// Mitsubishi GX Works2 project: auto0917   PLC: Q02/Q02H

PROGRAM MAIN
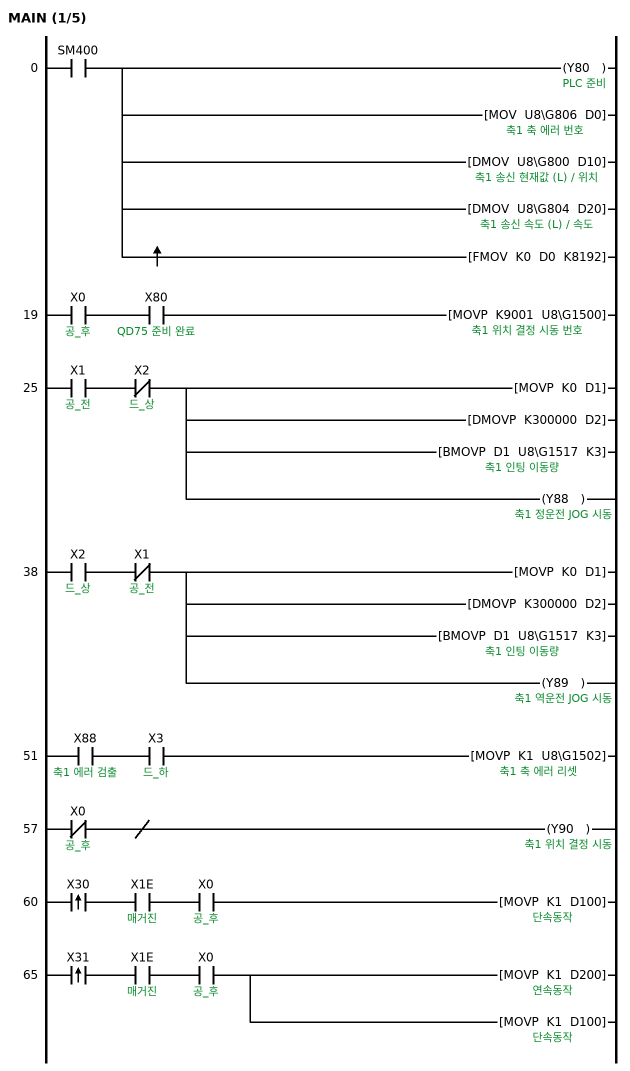
0     LD      SM400
      OUT     Y80  ; PLC 준비
      MOV     U8\G806 D0  ; 축1 축 에러 번호
      DMOV    U8\G800 D10  ; 축1 송신 현재값 (L) / 위치
      DMOV    U8\G804 D20  ; 축1 송신 속도 (L) / 속도
      MEP
      FMOV    K0 D0 K8192
19    LD      X0  ; 공_후
      AND     X80  ; QD75 준비 완료
      MOVP    K9001 U8\G1500  ; 축1 위치 결정 시동 번호
25    LD      X1  ; 공_전
      ANI     X2  ; 드_상
      MOVP    K0 D1
      DMOVP   K300000 D2
      BMOVP   D1 U8\G1517 K3  ; 축1 인팅 이동량
      OUT     Y88  ; 축1 정운전 JOG 시동
38    LD      X2  ; 드_상
      ANI     X1  ; 공_전
      MOVP    K0 D1
      DMOVP   K300000 D2
      BMOVP   D1 U8\G1517 K3
      OUT     Y89  ; 축1 역운전 JOG 시동
51    LD      X88  ; 축1 에러 검출
      AND     X3  ; 드_하
      MOVP    K1 U8\G1502  ; 축1 축 에러 리셋
57    LDI     X0  ; 공_후
      INV
      OUT     Y90  ; 축1 위치 결정 시동
60    LDP     X30
      AND     X1E  ; 매거진
      AND     X0  ; 공_후
      MOVP    K1 D100  ; 단속동작
65    LDP     X31
      AND     X1E  ; 매거진
      AND     X0  ; 공_후
      MOVP    K1 D200  ; 연속동작
      MOVP    K1 D100
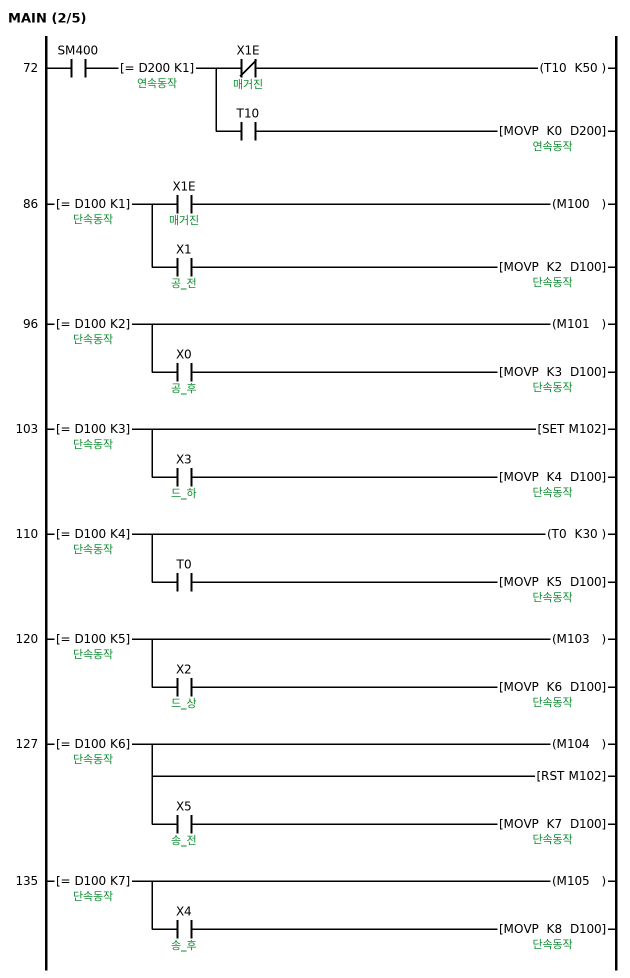
72    LD      SM400
      AND=    D200 K1  ; 연속동작
      MPS
      ANI     X1E  ; 매거진
      OUT     T10 K50
      MPP
      AND     T10
      MOVP    K0 D200
86    LD=     D100 K1  ; 단속동작
      MPS
      AND     X1E  ; 매거진
      OUT     M100
      MPP
      AND     X1  ; 공_전
      MOVP    K2 D100
96    LD=     D100 K2  ; 단속동작
      OUT     M101
      AND     X0  ; 공_후
      MOVP    K3 D100
103   LD=     D100 K3  ; 단속동작
      SET     M102
      AND     X3  ; 드_하
      MOVP    K4 D100
110   LD=     D100 K4  ; 단속동작
      OUT     T0 K30
      AND     T0
      MOVP    K5 D100
120   LD=     D100 K5  ; 단속동작
      OUT     M103
      AND     X2  ; 드_상
      MOVP    K6 D100
127   LD=     D100 K6  ; 단속동작
      OUT     M104
      RST     M102
      AND     X5  ; 송_전
      MOVP    K7 D100
135   LD=     D100 K7  ; 단속동작
      OUT     M105
      AND     X4  ; 송_후
      MOVP    K8 D100
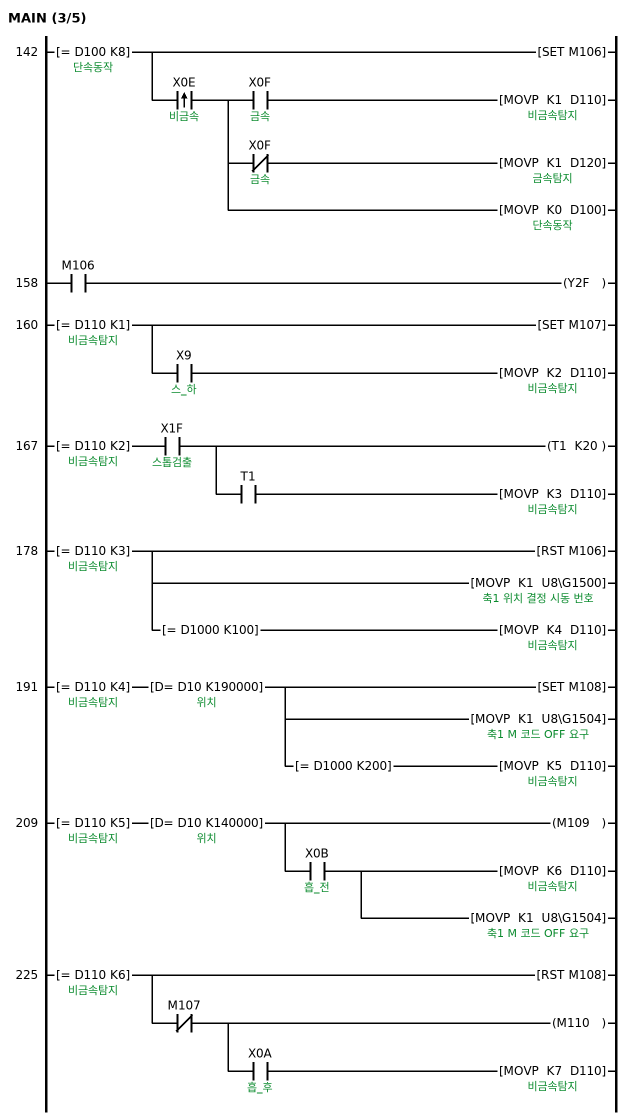
142   LD=     D100 K8  ; 단속동작
      SET     M106
      ANDP    X0E  ; 비금속
      MPS
      AND     X0F  ; 금속
      MOVP    K1 D110  ; 비금속탐지
      MRD
      ANI     X0F  ; 금속
      MOVP    K1 D120  ; 금속탐지
      MPP
      MOVP    K0 D100
158   LD      M106
      OUT     Y2F
160   LD=     D110 K1  ; 비금속탐지
      SET     M107
      AND     X9  ; 스_하
      MOVP    K2 D110
167   LD=     D110 K2  ; 비금속탐지
      AND     X1F  ; 스톱검출
      OUT     T1 K20
      AND     T1
      MOVP    K3 D110
178   LD=     D110 K3  ; 비금속탐지
      RST     M106
      MOVP    K1 U8\G1500
      AND=    D1000 K100
      MOVP    K4 D110
191   LD=     D110 K4  ; 비금속탐지
      ANDD=   D10 K190000  ; 위치
      SET     M108
      MOVP    K1 U8\G1504  ; 축1 M 코드 OFF 요구
      AND=    D1000 K200
      MOVP    K5 D110
209   LD=     D110 K5  ; 비금속탐지
      ANDD=   D10 K140000  ; 위치
      OUT     M109
      AND     X0B  ; 흡_전
      MOVP    K6 D110
      MOVP    K1 U8\G1504
225   LD=     D110 K6  ; 비금속탐지
      RST     M108
      ANI     M107
      OUT     M110
      AND     X0A  ; 흡_후
      MOVP    K7 D110
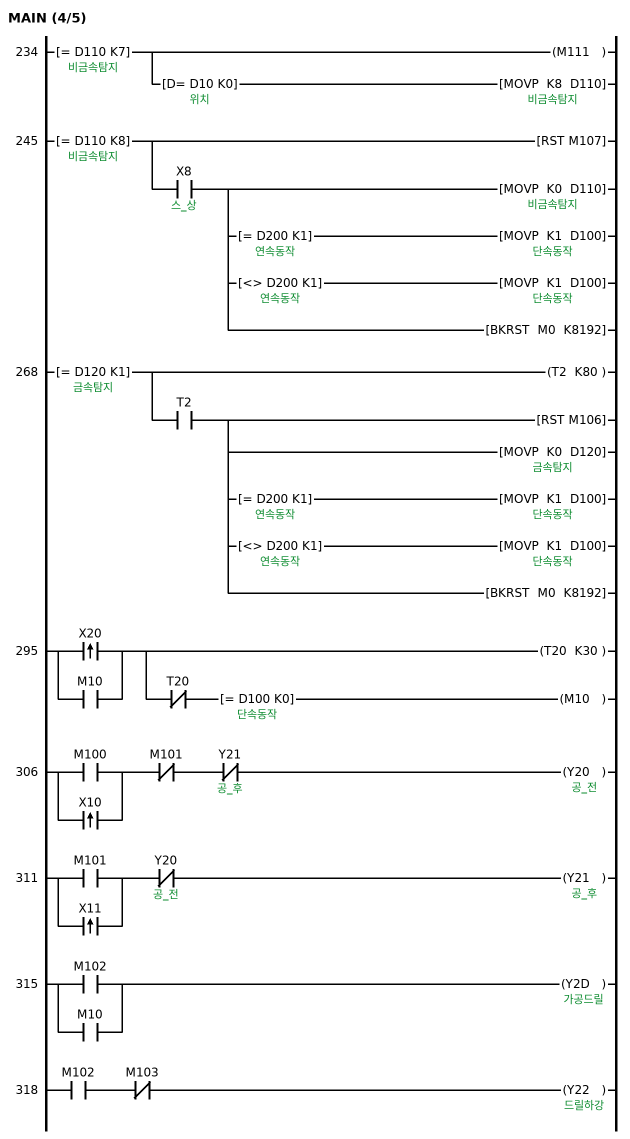
234   LD=     D110 K7  ; 비금속탐지
      OUT     M111
      ANDD=   D10 K0  ; 위치
      MOVP    K8 D110
245   LD=     D110 K8  ; 비금속탐지
      RST     M107
      AND     X8  ; 스_상
      MOVP    K0 D110
      MPS
      AND=    D200 K1  ; 연속동작
      MOVP    K1 D100
      MRD
      AND<>   D200 K1  ; 연속동작
      MOVP    K1 D100
      MPP
      BKRST   M0 K8192
268   LD=     D120 K1  ; 금속탐지
      OUT     T2 K80
      AND     T2
      RST     M106
      MOVP    K0 D120
      MPS
      AND=    D200 K1  ; 연속동작
      MOVP    K1 D100
      MRD
      AND<>   D200 K1  ; 연속동작
      MOVP    K1 D100
      MPP
      BKRST   M0 K8192
295   LDP     X20
      OR      M10
      OUT     T20 K30
      ANI     T20
      AND=    D100 K0  ; 단속동작
      OUT     M10
306   LD      M100
      ORP     X10
      ANI     M101
      ANI     Y21  ; 공_후
      OUT     Y20  ; 공_전
311   LD      M101
      ORP     X11
      ANI     Y20  ; 공_전
      OUT     Y21  ; 공_후
315   LD      M102
      OR      M10
      OUT     Y2D  ; 가공드릴
318   LD      M102
      ANI     M103
      OUT     Y22  ; 드릴하강
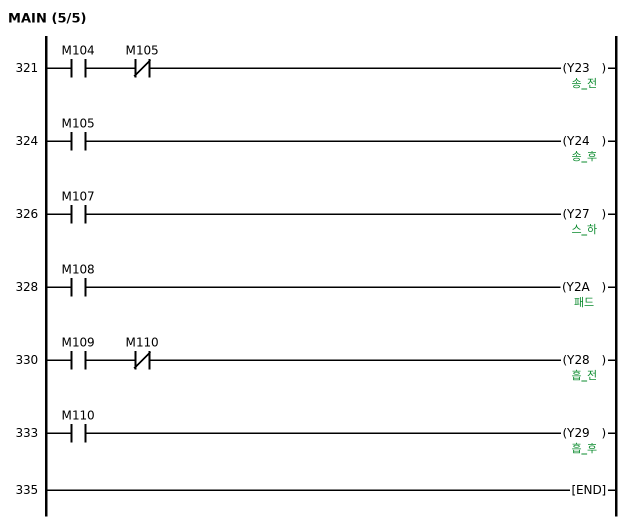
321   LD      M104
      ANI     M105
      OUT     Y23  ; 송_전
324   LD      M105
      OUT     Y24  ; 송_후
326   LD      M107
      OUT     Y27  ; 스_하
328   LD      M108
      OUT     Y2A  ; 패드
330   LD      M109
      ANI     M110
      OUT     Y28  ; 흡_전
333   LD      M110
      OUT     Y29  ; 흡_후
335   END
END_PROGRAM

PROGRAM MAIN1
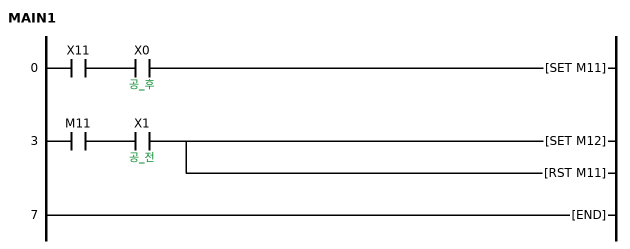
0     LD      X11
      AND     X0  ; 공_후
      SET     M11
3     LD      M11
      AND     X1  ; 공_전
      SET     M12
      RST     M11
7     END
END_PROGRAM

// device comments not shown above
X6  ; 배_후
X7  ; 배_전
X0C  ; 창_후
X0D  ; 창_전
X81  ; 동기용 플래그
X84  ; 축1 M 코드 ON
X85  ; 축2 M 코드 ON
X89  ; 축2 에러 검출
X8C  ; 축1 BUSY
X8D  ; 축2 BUSY
X90  ; 축1 시동 완료
X91  ; 축2 시동 완료
X94  ; 축1 위치 결정 완료
X95  ; 축2 위치 결정 완료
Y25  ; 배_전
Y26  ; 배_후
Y2B  ; 창_전
Y2C  ; 창_후
Y2E  ; 컨베이어
Y84  ; 축1 축 정지
Y85  ; 축2 축 정지
Y8A  ; 축2 정운전 JOG 시동
Y8B  ; 축2 역운전 JOG 시동
Y91  ; 축2 위치 결정 시동
Y94  ; 축1 실행 금지 플래그
Y95  ; 축2 실행 금지 플래그
